// TIA Portal V20 export
TYPE "posSetpoint"
// stored: Access Published, Namespace Unit1
   STRUCT
      "Postive PV" : LReal;
      "Negative PV" : LReal;
      "Set Pos" : LReal;
      inPos : Bool;
      isBefore : Bool;
      isAfter : Bool;
   END_STRUCT;
END_TYPE
